// ---- POUs/UNIT/fb_Clamp/FB_ClampMove.TcPOU
FUNCTION_BLOCK FB_ClampMove
VAR_INPUT
	Ex	:BOOL;
	UnitMode	:DINT;
	paraAutoMove		:INT;
	_iHeavyGauge: INT;
END_VAR
VAR_OUTPUT
	Done	:BOOL;
END_VAR
VAR
	inMid,inFrnt,inRear,inMid2: INPUT;
	
	tonDone: Ton;
	aa: BOOL;
	iStep: INT;
	ton11: ton;
END_VAR

(*-----------------------------------------------------------------------------------*)
(*------------------------- Clamp Gauge Front/Rear/Middle ---------------------------*)
(*-----------------------------------------------------------------------------------*)


inMid(PT_OFF:=T#3S );
inFrnt(PT_OFF:=T#3S );
inRear(PT_OFF:=T#3S );
inMid2(PT_OFF:=T#3S );
CASE iStep OF
	0:
		IF stFolder.Status.Clamp_GtLowPoint AND Ex THEN
			iStep:=1;
		END_IF
	1:
	inMid.INPUT		:=Hmi_bArray[1] AND NOT In_sigGaugingMid;		//Light 			
	inFrnt.INPUT	:=NOT Hmi_bArray[1] AND _iHeavyGauge=+1 AND (NOT In_sigGaugingFrnt);//Heavy
	inRear.INPUT	:=NOT Hmi_bArray[1] AND _iHeavyGauGE=-1 AND (NOT In_sigGaugingRear);//Heavy
	inMid2.INPUT	:=NOT Hmi_bArray[1] AND _iHeavyGauGE=0  AND (NOT In_sigGaugingMid);	//Heavy Sqlusa
	IF (Hmi_bArray[1] AND In_sigGaugingMid) OR 
		(NOT Hmi_bArray[1] AND _iHeavyGauge=+1 AND In_sigGaugingFrnt) OR
		(NOT Hmi_bArray[1] AND _iHeavyGauge=-1 AND In_sigGaugingRear) OR
		(NOT Hmi_bArray[1] AND _iHeavyGauge= 0 AND In_sigGaugingMid) THEN
		iStep:=2;
	END_IF
	2:
	iStep:=3;
	3:
	iStep:=4;
	4:
	iStep:=5;
	5:
	IF NOT inFrnt.Q AND NOT inRear.Q AND NOT inMid.Q AND NOT inMid2.Q  THEN
		iStep:=10;
	END_IF
	10:
	Out_GaugingF_Ext:=Out_GaugingF_Rtn:=Out_GaugingR_Ext:=Out_GaugingR_Rtn:=FALSE;
	ton11(IN:=TRUE , PT:=T#300MS , Q=> , ET=> );
	IF ton11.Q THEN
		iStep:=11;
	END_IF
	11:
	ton11(IN:=FALSE );
	
	Done	:=TRUE;
	iStep:=0;
	Ex	:=FALSE;
	
END_CASE


	
//上钳口工作位：若Front信号未到，一直输出Front阀。直到Front信号到，延时1秒后，关闭阀。

IF inMid.Q OR inMid2.Q THEN
	Out_GaugingF_Ext:=TRUE;		Out_GaugingF_Rtn:=FALSE;	Out_GaugingR_Ext:=FALSE;	Out_GaugingR_Rtn:=TRUE;		//Middle 0mm
ELSIF inFrnt.Q THEN
	Out_GaugingF_Ext:=TRUE;		Out_GaugingF_Rtn:=FALSE;	Out_GaugingR_Ext:=TRUE;		Out_GaugingR_Rtn:=FALSE;		//Front +2MM
ELSIF inRear.Q THEN
	Out_GaugingF_Ext:=FALSE; 	Out_GaugingF_Rtn:=TRUE;		Out_GaugingR_Ext:=FALSE;	Out_GaugingR_Rtn:=TRUE;			//Rear -2MM

	
END_IF

	

tonDone(IN:=Done , PT:=T#2000MS , Q=> , ET=> );
IF tonDone.Q THEN
	Done	:=FALSE;
	
END_IF

END_FUNCTION_BLOCK

// ---- VISUs/VISUs/Templates/VIS_TemplateCommand.TcVIS
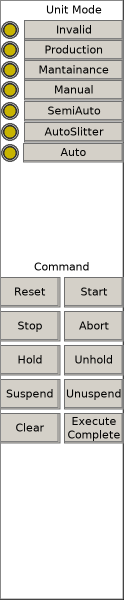
VISUALIZATION VIS_TemplateCommand  // 124x600
VAR_IN_OUT
	eModeCommand	: DINT;
	eStateCommand	: DINT;
	eModeStatus		: DINT;
	eStateStatus	: DINT;
	bModeChangeReq	: BOOL;
END_VAR
    Rectangle (0,0 124x600)
    Lamp1 (0,20 20x20), variable: (eModeStatus = 0), style: Lamp-Lamp1-Yellow
    Button (24,20 100x20), "Invalid", colour toggle: (eModeStatus = 0)
        tap bModeChangeReq
        OnMouseClick: execute { eModeCommand := 0; }
    Lamp1 (0,40 20x20), variable: (eModeStatus = 1), style: Lamp-Lamp1-Yellow
    Button (24,40 100x20), "Production"
        tap bModeChangeReq
        OnMouseClick: execute { eModeCommand := 1; }
    Lamp1 (0,60 20x20), variable: (eModeStatus = 2), style: Lamp-Lamp1-Yellow
    Button (24,60 100x20), "Mantainance"
        tap bModeChangeReq
        OnMouseClick: execute { eModeCommand := 2; }
    Lamp1 (0,80 20x20), variable: (eModeStatus = 3), style: Lamp-Lamp1-Yellow
    Button (24,80 100x20), "Manual"
        tap bModeChangeReq
        OnMouseClick: execute { eModeCommand := 3; }
    Button (0,277 60x30), "Reset"
        OnMouseClick: execute { eStateCommand := 1; }
    Button (64,277 60x30), "Start"
        OnMouseClick: execute { eStateCommand := 2; }
    Button (0,311 60x30), "Stop"
        OnMouseClick: execute { eStateCommand := 3; }
    Button (0,345 60x30), "Hold"
        OnMouseClick: execute { eStateCommand := 4; }
    Button (64,345 60x30), "Unhold"
        OnMouseClick: execute { eStateCommand := 5; }
    Button (0,379 60x30), "Suspend"
        OnMouseClick: execute { eStateCommand := 6; }
    Button (64,379 60x30), "Unuspend"
        OnMouseClick: execute { eStateCommand := 7; }
    Button (0,413 60x30), "Clear"
        OnMouseClick: execute { eStateCommand := 9; }
    Label (0,257 124x20), "Command"
    Button (64,311 60x30), "Abort"
        OnMouseClick: execute { eStateCommand := 8; }
    Button (64,413 60x30), "Execute Complete"
        OnMouseClick: execute { MAIN.bExecuteComplete := TRUE; }
    Label (24,0 100x20), "Unit Mode"
    Button (24,101 100x20), "SemiAuto"
        tap bModeChangeReq
        OnMouseClick: execute { eModeCommand := 4; }
    Lamp1 (0,101 20x20), variable: (eModeStatus = 4), style: Lamp-Lamp1-Yellow
    Button (24,122 100x20), "AutoSlitter"
        tap bModeChangeReq
        OnMouseClick: execute { eModeCommand := 5; }
    Lamp1 (0,122 20x20), variable: (eModeStatus = 5), style: Lamp-Lamp1-Yellow
    Button (23,143 101x19), "Auto"
        tap bModeChangeReq
        OnMouseClick: execute { eModeCommand := 6; }
    Lamp1 (0,143 20x20), variable: (eModeStatus = 6), style: Lamp-Lamp1-Yellow
END_VISUALIZATION

// ---- VISUs/VISUs/VIS_Main.TcVIS
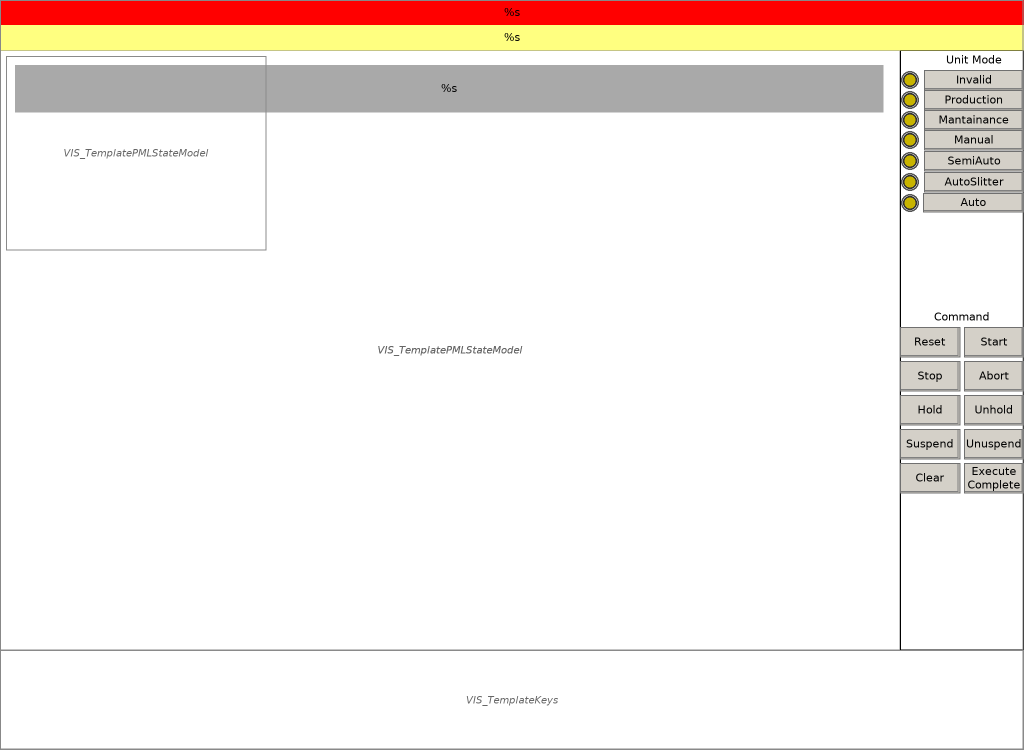
VISUALIZATION VIS_Main  // 1024x750
    Frame (0,50 900x600), invisible if: MAIN.fbVisu.iFrameVisible = 0 OR MAIN.fbMachine.bChangeIntoProduction
        shows VIS_TemplatePMLStateModel(ePMLUnitMode := MAIN.fbVisu.eModeVisu, ePMLState := MAIN.fbVisu.eStateVisu)
    Textfield (15,65 868x47), "%s", text variable: MAIN.fbVisu.sUnitName, invisible if: MAIN.fbVisu.iFrameVisible = 0 OR MAIN.fbMachine.bChangeIntoProduction
    Frame (0,50 900x600), invisible if: MAIN.fbVisu.iFrameVisible > 0 OR MAIN.fbMachine.bChangeIntoProduction
        shows VIS_TemplatePMLStateModel(ePMLUnitMode := MAIN.fbVisu.eModeVisu, ePMLState := MAIN.fbVisu.eStateVisu)
    Rectangle (0,0 1024x25), "%s", text variable: MAIN.fbVisu.sAlarmVisu, invisible if: (MAIN.fbMachine.bChangeIntoProduction OR MAIN.fbVisu.sAlarmVisu = '')
    Frame (900,50 124x600)
        shows VIS_TemplateCommand(eModeCommand := PackTags.Command.UnitMode, eStateCommand := PackTags.Command.CntrlCmd, eModeStatus := PackTags.Status.UnitModeCurrent, eStateStatus := PackTags.Status.StateCurrent, bModeChangeReq := PackTags.Command.UnitModeChangeRequest)
    Frame (0,650 1024x100)
        shows VIS_TemplateKeys(Caption := aCaption, KeyPressed := aKeyPressed)
    Frame (6,56 260x194), invisible if: MAIN.fbVisu.iFrameVisible > 0 OR MAIN.fbMachine.bChangeIntoProduction
        shows VIS_TemplatePMLStateModel(ePMLUnitMode := PackTags.Status.UnitModeCurrent, ePMLState := PackTags.Status.StateCurrent)
    Rectangle (0,25 1024x25), "%s", text variable: MAIN.fbVisu.sWarningVisu, invisible if: (MAIN.fbMachine.bChangeIntoProduction OR MAIN.fbVisu.sWarningVisu ='')
END_VISUALIZATION
